TYPE ST_LIST_CTRL :
STRUCT
  Cmd         : E_LIST_CTRL;
END_STRUCT
END_TYPE

(* stored: Version 1.1.0.1, ProductVersion 3.1.4026.18
   DUT ST_LIST_CTRL: Id {b4557692-394b-48bc-85bb-4dacfd26bb20} *)
